{attribute 'qualified_only'}
{attribute 'strict'}
TYPE DiscretizationType :
(
  Continuous, /// Every trajectory synchronization duration is allowed (Default)
  Discrete /// The trajectory synchronization duration must be a multiple of the control cycle
);
END_TYPE

(* stored: Version 1.1.0.1
   DUT DiscretizationType: Id {57780566-a3c2-481a-ac6d-a6d55abca32c} *)
